// TwinCAT 3 PLC project SIM
// ProgramVersion: 3.1.4026.22
// libraries:
//   Tc2_Standard, * (Beckhoff Automation GmbH)
//   Tc2_System, * (Beckhoff Automation GmbH)
// project tree:
//   / PlcTask.TcTTO
//   POUs/ MAIN.TcPOU, F_Noise.TcPOU, F_Random.TcPOU
// (motion and I/O tree: see PLC project plc)
// real-time tasks:
//   TASK PlcTask: cycle T#10ms, priority 20, ADS port 350
//   TASK PlcTask1: cycle T#10ms, priority 21, ADS port 351
// variable links:
//   PLC/PLC Instance <-> SIM/SIM Instance
//     PlcTask Inputs/MAIN.bCycleRun <-> PlcTask Outputs/MAIN.bCycleRun
//     PlcTask Inputs/MAIN.fMotorCurrent <-> PlcTask Outputs/MAIN.fMotorCurrent
//     PlcTask Inputs/MAIN.fTemperature <-> PlcTask Outputs/MAIN.fTemperature
//     PlcTask Inputs/MAIN.fVibration <-> PlcTask Outputs/MAIN.fVibration
//     PlcTask Inputs/MAIN.nCycleTime <-> PlcTask Outputs/MAIN.nCycleTimeActual

CONFIGURATION SIM
    RESOURCE PLC ON TwinCAT3
        TASK PlcTask(INTERVAL := T#10ms, PRIORITY := 21);
        PROGRAM MAIN WITH PlcTask : MAIN;
    END_RESOURCE
END_CONFIGURATION

// ---- POUs/MAIN.TcPOU
PROGRAM MAIN
VAR
	bStart				: BOOL := TRUE;
	
	fMotorCurrent		AT %Q* : LREAL;
	fTemperature		AT %Q* : LREAL;
	fVibration			AT %Q* : LREAL;
	nCycleTimeActual	AT %Q* : DINT;
	bCycleRun			AT %Q* : BOOL;
	
	nScanCount			: DINT;
	nCycleLength		: DINT;
	nIdleLength			: DINT;
	nState				: DINT;
	fBaseLoad			: LREAL;
	fLoad				: LREAL;
	fTnorm				: LREAL;
	
	fWearItem			: LREAL := 0.001;
	nTempCycles			: DINT;
	fTempFactor			: LREAL;
	
END_VAR

CASE nState OF
	0:
		// idle
		IF bStart THEN
			nState := 1;
		END_IF
	1:
		bCycleRun := FALSE;
	
		// Idle signals (baseline)
		fTemperature := 32.0 + F_Noise(0.01) + (TO_LREAL(nTempCycles) / 50.0);
		fVibration  := 0.01 + F_Noise(0.01);
		fMotorCurrent := 2.0 + F_Noise(0.1);
	
		nScanCount := nScanCount + 1;

		IF nScanCount >= nIdleLength THEN
			// Start new cycle
			nState := 2;
			nScanCount := 0;
	
			nCycleLength := 25;
			nIdleLength := 100;
	
			// Slight load variation
			fBaseLoad := fBaseLoad + (F_Random() - 0.5) * 0.05;
			fBaseLoad := LIMIT(0.3, fBaseLoad, 1.0);
		END_IF
	
	2:
		bCycleRun := TRUE;
	
		// Normalized time (0 → 1)
		fTnorm := TO_LREAL(nScanCount) / TO_LREAL(nCycleLength);
	
		// -------------------------
		// Load profile
		// -------------------------
		IF fTnorm < 0.2 THEN
			fLoad := fBaseLoad * (fTnorm / 0.2);
		ELSIF fTnorm < 0.8 THEN
			fLoad := fBaseLoad;
		ELSE
			fLoad := fBaseLoad * (1.0 - (fTnorm - 0.8) / 0.2);
		END_IF
	
		// -------------------------
		// Signal generation
		// -------------------------
	
		fVibration := 0.2
			+ (fLoad * 2.5)
			+ (fWearItem * 5.0)
			+ (fTempFactor * 2.0)
			+ F_Noise(0.5 + (fWearItem * 2.5) + fTempFactor);
	
		fMotorCurrent := 5.0
			+ (fLoad * 10.0)
			+ (fWearItem * 4.0)
			+ F_Noise(0.2 + fWearItem + (fTempFactor * 1.25));
			
		nCycleTimeActual := 210 + TO_DINT(F_Random() * 25);
	
		// -------------------------
		// Advance time
		// -------------------------
		nScanCount := nScanCount + 1;
	
		IF nScanCount >= nCycleLength THEN
			// End cycle
			nState := 1;
			nScanCount := 0;
			
			IF fWearItem < 0.25 THEN
				fWearItem := fWearItem + (F_Random() / 300);
			ELSE
				fWearItem := 0.001;
			END_IF
	
			IF F_Random() < 0.01 THEN
				nTempCycles := 0;
			ELSE
				nTempCycles := nTempCycles + (225 - nCycleTimeActual);
			END_IF
			
			fTempFactor := (fTemperature - 32.0) / 4.0;
			
			// Clear fault sometimes
			(*IF RANDOM() < 0.5 THEN
				faultActive := FALSE;
			END_IF
	
			// Increase wear slowly
			wear := wear + 0.002;
			LIMIT(wear, 0.0, 1.0);*)
		END_IF
	
END_CASE

END_PROGRAM

// ---- POUs/F_Noise.TcPOU
FUNCTION F_Noise : LREAL
VAR_INPUT
	fAmplitude		: LREAL;
END_VAR
VAR
	fR				: LREAL;
END_VAR

fR := (F_Random() + F_Random() + F_Random()) / 3.0;
fR := (fR * 2.0) - 1.0;
F_Noise := fR * fAmplitude;

END_FUNCTION

// ---- POUs/F_Random.TcPOU
FUNCTION F_Random : LREAL
VAR_INPUT
END_VAR
VAR
	nSeed 		: INT;
	rand		: DRAND;
	fbCpu		: GETCPUCOUNTER;
	nLow		: DWORD;
END_VAR

fbCpu(cpuCntLoDW => nLow);
nSeed := TO_INT(nLow);
rand(Seed:=nSeed);
F_Random := rand.Num;

END_FUNCTION
